// TIA Portal V17 export
// export: Created 2023-04-03T06:31:41.664051Z, ExportSetting WithDefaults, DisplayName Totally Integrated Automation Portal, DisplayVersion V17 Update 4, DisplayName TIA Portal Openness, DisplayVersion V17 Update 4, DisplayName TIA Portal Version Control Interface, DisplayVersion V17, DisplayName STEP 7 Professional, DisplayVersion V17 Update 4, DisplayName STEP 7 Safety, DisplayVersion V17, DisplayName WinCC Professional, DisplayVersion V17 Update 4
TYPE "CATL_CELL_V"
// stored: IsFailsafeCompliant false
   STRUCT
      CSC_Volt_Cell1 : Real;
      CSC_Volt_Cell2 : Real;
      CSC_Volt_Cell3 : Real;
      CSC_Volt_Cell4 : Real;
      CSC_Volt_Cell5 : Real;
      CSC_Volt_Cell6 : Real;
      CSC_Volt_Cell7 : Real;
      CSC_Volt_Cell8 : Real;
      CSC_Volt_Cell9 : Real;
      CSC_Volt_Cell10 : Real;
      CSC_Volt_Cell11 : Real;
      CSC_Volt_Cell12 : Real;
      CSC_Volt_Cell13 : Real;
      CSC_Volt_Cell14 : Real;
      CSC_Volt_Cell15 : Real;
      CSC_Volt_Cell16 : Real;
      CSC_Volt_Cell17 : Real;
      CSC_Volt_Cell18 : Real;
      CSC_Volt_Cell19 : Real;
      CSC_Volt_Cell20 : Real;
      CSC_Volt_Cell21 : Real;
      CSC_Volt_Cell22 : Real;
      CSC_Volt_Cell23 : Real;
      CSC_Volt_Cell24 : Real;
      CSC_Volt_Cell25 : Real;
      CSC_Volt_Cell26 : Real;
      CSC_Volt_Cell27 : Real;
      CSC_Volt_Cell28 : Real;
      CSC_Volt_Cell29 : Real;
      CSC_Volt_Cell30 : Real;
      CSC_Volt_Cell31 : Real;
      CSC_Volt_Cell32 : Real;
      CSC_Volt_Cell33 : Real;
      CSC_Volt_Cell34 : Real;
      CSC_Volt_Cell35 : Real;
      CSC_Volt_Cell36 : Real;
      CSC_Volt_Cell37 : Real;
      CSC_Volt_Cell38 : Real;
      CSC_Volt_Cell39 : Real;
      CSC_Volt_Cell40 : Real;
      CSC_Volt_Cell41 : Real;
      CSC_Volt_Cell42 : Real;
      CSC_Volt_Cell43 : Real;
      CSC_Volt_Cell44 : Real;
      CSC_Volt_Cell45 : Real;
      CSC_Volt_Cell46 : Real;
      CSC_Volt_Cell47 : Real;
      CSC_Volt_Cell48 : Real;
      CSC_Volt_Cell49 : Real;
      CSC_Volt_Cell50 : Real;
      CSC_Volt_Cell51 : Real;
      CSC_Volt_Cell52 : Real;
   END_STRUCT;
END_TYPE
